Fanuc KAREL source: POS2JOINT.kl

PROGRAM T
%NOLOCKGROUP
VAR
 v0 : JOINTPOS
 v1 : POSITION
 v2 : POSITION
 v3 : POSITION
 v4 : INTEGER
 v5 : CONFIG
 v6 : ARRAY[10] OF REAL
 v7 : JOINTPOS
 v8 : INTEGER
BEGIN
 POS2JOINT(v0, v1, v2, v3, v4, v5, v6, v7, v8)
END T
